FUNCTION MSG_CONCAT : STRING(3500)
VAR_INPUT
	_DeviceState : ARRAY[1..14] OF DeviceAttr;
	_SystemTime	 : STRING;
END_VAR
VAR
	API_JSON		: ARRAY[1..14] OF STRING(255);
	index			: INT;
	success			: BOOL;
	API_MSG			: STRING(3500);
	sopenBracket	: STRING(13) := '{"dbLists":[';
END_VAR


//success := CONCAT2(pSrcString1 := ADR(_text), pSrcString2 := ADR(_SystemTime), pDstString := ADR(API_JSON), nDstSize := SIZEOF(API_JSON));

FOR index:=1 TO 14 DO 
	API_JSON[index] := CONCAT(API_JSON[index],'{"ObjectData":{"ObjectId":"');	
	API_JSON[index] := CONCAT(API_JSON[index],_DeviceState[index].DeviceID);
	API_JSON[index] := CONCAT(API_JSON[index],'","ActionData":[{"Key":"');
	API_JSON[index] := CONCAT(API_JSON[index],_DeviceState[index].ActionKey);
	API_JSON[index] := CONCAT(API_JSON[index],'","Value":"');
	API_JSON[index] := CONCAT(API_JSON[index],USINT_TO_STRING(_DeviceState[index].ActionVal));
	API_JSON[index] := CONCAT(API_JSON[index],'","TimeStamp":');
	API_JSON[index] := CONCAT(API_JSON[index],_SystemTime);
	API_JSON[index] := CONCAT(API_JSON[index],'}],"Attributes":[{"Key":"');
	API_JSON[index] := CONCAT(API_JSON[index],_DeviceState[index].OnlineKey);
	API_JSON[index] := CONCAT(API_JSON[index],'","Value":"');
	API_JSON[index] := CONCAT(API_JSON[index],USINT_TO_STRING(_DeviceState[index].OnlineVal));
	API_JSON[index] := CONCAT(API_JSON[index],'","TimeStamp":');
	API_JSON[index] := CONCAT(API_JSON[index],_SystemTime);
	API_JSON[index] := CONCAT(API_JSON[index],'},{"Key":"');
	API_JSON[index] := CONCAT(API_JSON[index],_DeviceState[index].ErrorKey);
	API_JSON[index] := CONCAT(API_JSON[index],'","Value":"');
	API_JSON[index] := CONCAT(API_JSON[index],USINT_TO_STRING(_DeviceState[index].ErrorVal));
	API_JSON[index] := CONCAT(API_JSON[index],'","TimeStamp":');
	API_JSON[index] := CONCAT(API_JSON[index],_SystemTime);
	IF index < 14 THEN
		API_JSON[index] := CONCAT(API_JSON[index],'}]}},');
	ELSE
		API_JSON[index] := CONCAT(API_JSON[index],'}]}}]}');
	END_IF
	success := CONCAT2(pSrcString1 := ADR(API_MSG), pSrcString2 := ADR(API_JSON[index]), pDstString := ADR(API_MSG), nDstSize := SIZEOF(API_MSG));
END_FOR
	success := CONCAT2(pSrcString1 := ADR(sopenBracket), pSrcString2 := ADR(API_MSG), pDstString := ADR(API_MSG), nDstSize := SIZEOF(API_MSG));
MSG_CONCAT := API_MSG;

END_FUNCTION

(* stored: Version 1.1.0.1, ProductVersion 3.1.4024.12
   POU MSG_CONCAT: Id {dcfa6f3e-ed15-4c3f-afbb-ab1a1d0281a7}, SpecialFunc None *)
